FUNCTION_BLOCK OutputPorts Implements I_OutputPorts
VAR
	ports : Stack;
END_VAR

METHOD PUBLIC GetEnumerator : I_ForwardEnumerator
VAR_INPUT
END_VAR
GetEnumerator := ports.GetEnumerator();
END_METHOD

METHOD PUBLIC Insert
VAR_INPUT
	PortToInsert : I_OutputPort;
END_VAR
ports.Push(PortToInsert);
END_METHOD

METHOD PUBLIC TryGetByName : BOOL
VAR_INPUT
	Name : STRING;
	Destination : REFERENCE TO I_OutputPort;
END_VAR
VAR
	portEnumerator : I_ForwardEnumerator;
	port : I_OutputPort;
END_VAR
portEnumerator := ports.GetEnumerator();

WHILE portEnumerator.MoveNext() DO 
	IF  NOT portEnumerator.TryGet(port) THEN
		CONTINUE;
	END_IF
	
	IF port.Name = Name THEN 
		TryGetByName := TRUE;
		Destination := port;
		EXIT;
	END_IF

END_WHILE

portEnumerator.Dispose();
END_METHOD

END_FUNCTION_BLOCK

(* stored: Version 1.1.0.1, ProductVersion 3.1.4024.12
   POU OutputPorts: Id {9694add8-d5ac-0816-0153-5912f1890314}, SpecialFunc None
   Method GetEnumerator: Id {040b39cf-2e50-0b84-217b-6135200fce42}
   Method Insert: Id {9fec9190-707f-0a99-2132-8f3742ae5ba6}
   Method TryGetByName: Id {25a107fc-d85c-0e84-108a-c9a721c8bdc5} *)
